// Mitsubishi GX Works2 project: main   PLC: Q02/Q02H

// task Task_01 (event TRUE, interval 0, priority 31): POU_01

PROGRAM POU_01
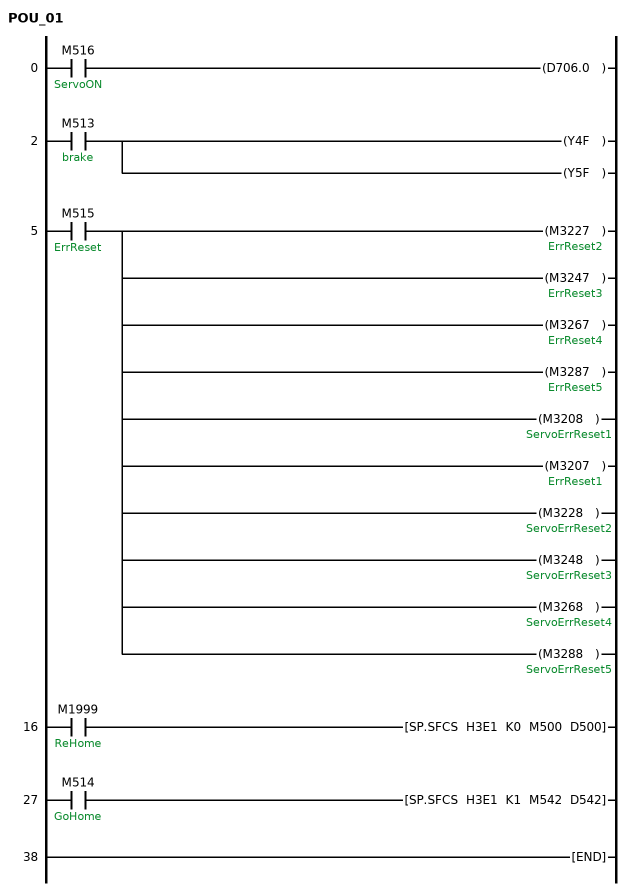
0     LD      M516  ; ServoON
      OUT     D706.0
2     LD      M513  ; brake
      OUT     Y4F
      OUT     Y5F
5     LD      M515  ; ErrReset
      OUT     M3227  ; ErrReset2
      OUT     M3247  ; ErrReset3
      OUT     M3267  ; ErrReset4
      OUT     M3287  ; ErrReset5
      OUT     M3208  ; ServoErrReset1
      OUT     M3207  ; ErrReset1
      OUT     M3228  ; ServoErrReset2
      OUT     M3248  ; ServoErrReset3
      OUT     M3268  ; ServoErrReset4
      OUT     M3288  ; ServoErrReset5
16    LD      M1999  ; ReHome
      SP.SFCS H3E1 K0 M500 D500
27    LD      M514  ; GoHome
      SP.SFCS H3E1 K1 M542 D542
38    END
END_PROGRAM

// device comments not shown above
M512  ; PLC ready flag request
M517  ; p2p
M519  ; modbus
M520  ; conveyor
M521  ; reset
M522  ; runman
M526  ; symetric
M536  ; writeRS232
M537  ; readRS232
M543  ; position
M544  ; speed
M1000  ; Accep flag 1
M1001  ; Accep flag 2
M1002  ; Accep flag 3
M1003  ; Accep flag 4
M1004  ; Accep flag 5
M1005  ; Servo ready 1
M1006  ; Servo ready 2
M1007  ; Servo ready 3
M1008  ; Servo ready 4
M1009  ; Servo ready 5
M1010  ; Error 1
M1011  ; Error 2
M1012  ; Error 3
M1013  ; Error 4
M1014  ; Error 5
M1015  ; ready flag
M1016  ; brake
M1987  ; reset
M1988  ; conveyor
M1989  ; symetric
M1993  ; manrun
M1994  ; modbus
M1995  ; runall
M1997  ; moveJog
M1998  ; ReHome
M2000  ; PLC Ready flag
M2001  ; StartAceptFlag1
M2002  ; StartAceptFlag2
M2003  ; StartAceptFlag3
M2004  ; StartAceptFlag4
M2005  ; StartAceptFlag5
M2407  ; ErrDetec1
M2408  ; SerErrDetec1
M2415  ; ServoReady1
M2427  ; ErrDetec2
M2428  ; SerErrDetec2
M2435  ; ServoReady2
M2447  ; ErrDetec3
M2448  ; SerErrDetec3
M2455  ; ServoReady3
M2467  ; ErrDetec4
M2468  ; SerErrDetec4
M2475  ; ServoReady4
M2487  ; ErrDetec5
M2488  ; SerErrDetec5
M2495  ; ServoReady5
M3840  ; SFC flag
M3842  ; get camera
M3843  ; Run Only
M3844  ; gang tay
Y4E  ; gripper
D0  ; FeedCVal1
D20  ; FeedCVal2
D40  ; FeedCVal3
D60  ; FeedCVal4
D80  ; FeedCVal5
D704  ; PLC ready flag request
D705  ; passpoint
D706  ; ServoON
D859  ; run
D2010  ; addresspoint1
D2012  ; addresspoint2
D2014  ; addresspoint3
D2016  ; addresspoint4
D2018  ; addresspoint5
D10302  ; No.Protocol
D10320  ; slaveID
D10321  ; address
D10322  ; No.Resister
T0  ; timer out
